PROGRAM P_Demo_FB_HVACWork
VAR
    fb : FB_HVACWork;                            // 被演示 FB 实例
    eDataSecurityType_in : E_HVACDataSecurityType ;
    bSetDefault_in : BOOL := FALSE;
    bOn_in : BOOL := FALSE;
    bResetHours_in : BOOL := FALSE;
    bResetCount_in : BOOL := FALSE;
    dtSystemtime_in : DT ;
    bStartWarnLevel_in : BOOL := FALSE;
    bStartAlarmLevel_in : BOOL := FALSE;
    bSysTakt1Hz_in : BOOL := FALSE;
    bReset_in : BOOL := FALSE;
    rHours_io : REAL := 0.0;
    uiCount_io : UINT := 0;
    uiWarnLevel_io : UINT := 0;
    uiAlarmLevel_io : UINT := 0;
    bEnableWarnLevel_io : BOOL := FALSE;
    bEnableAlarmLevel_io : BOOL := FALSE;
    bQAlarmLevel_out : BOOL;
    bQWarnLevel_out : BOOL;
    bInvalidParameter_out : BOOL;
END_VAR

// ============================================================================
// Tc2_HVAC.FB_HVACWork 演示程序
// ============================================================================
// 场景：把本 FB 实例化到一个 PLC 程序里，每周期单次调用；按需要把 VAR_INPUT 与
//       VAR_IN_OUT 接到工程信号；VAR_OUTPUT 写入对应监视变量。
// 价值：使用本 FB 比手写状态机 / 控制算法节省大量代码；与 Tc2_HVAC 体系内其它 FB
//       直接对接，命名 / 持久化 / 模式仲裁等约定一致。具体语义见 FB_HVACWork.md 主文档。
// 验证步骤：
//   1. 右键 PLC 项目下 POUs 文件夹 → Add → Existing Item → 选本 .TcPOU 文件
//   2. 引用 Tc2_HVAC（References → Add library）
//   3. 编译 → 登录 → 运行
//   4. 在线写各 *_in 输入信号触发 FB；在线 monitor *_out 引脚观察状态
// ============================================================================

fb(
    eDataSecurityType := eDataSecurityType_in,
    bSetDefault := bSetDefault_in,
    bOn := bOn_in,
    bResetHours := bResetHours_in,
    bResetCount := bResetCount_in,
    dtSystemtime := dtSystemtime_in,
    bStartWarnLevel := bStartWarnLevel_in,
    bStartAlarmLevel := bStartAlarmLevel_in,
    bSysTakt1Hz := bSysTakt1Hz_in,
    bReset := bReset_in,
    rHours := rHours_io,
    uiCount := uiCount_io,
    uiWarnLevel := uiWarnLevel_io,
    uiAlarmLevel := uiAlarmLevel_io,
    bEnableWarnLevel := bEnableWarnLevel_io,
    bEnableAlarmLevel := bEnableAlarmLevel_io,
    bQAlarmLevel => bQAlarmLevel_out,
    bQWarnLevel => bQWarnLevel_out,
    bInvalidParameter => bInvalidParameter_out
);

END_PROGRAM

(* stored: Version 1.1.0.1, ProductVersion 3.1.4024.5
   POU P_Demo_FB_HVACWork: Id {418bca30-c672-5b46-8f0a-5655a410f7ab}, SpecialFunc None *)
